Omron CX-Programmer project NewProject (CX-Programmer 9.61)

# PLC NewPLC1: CP1E N30

## Global symbols (name address type ; comment)
0.00 BOOL  ; PB1
0.01 BOOL  ; LS1
0.02 BOOL  ; PS1
0.03 BOOL  ; SS1
0.04 BOOL  ; LS2
0.05 BOOL  ; LS3
0.06 BOOL  ; PB2
0.07 BOOL  ; PB3
0.08 BOOL  ; LS4
100.00 BOOL  ; CR1
100.01 BOOL  ; PL1
100.02 BOOL  ; SOLA
100.03 BOOL  ; CR2
100.04 BOOL  ; SOLB
100.05 BOOL  ; SOLC
100.06 BOOL  ; CR3
100.07 BOOL  ; PL2

## Program NewProgram1 (cyclic task 0)

### Section Section1

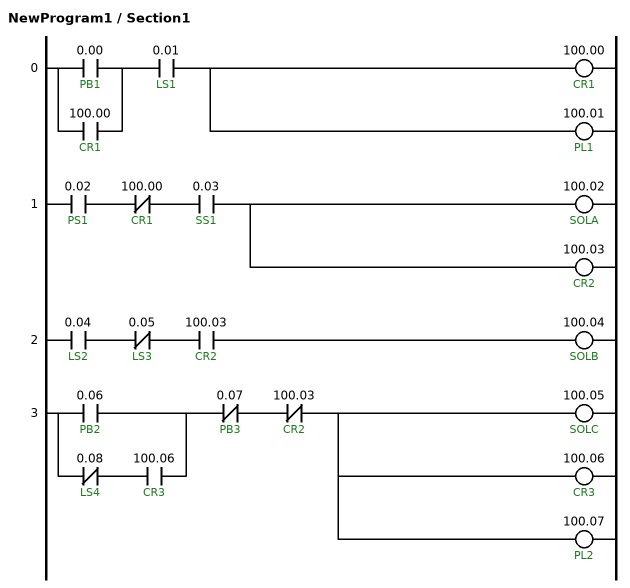
; rung 0
LD 0.00  ; PB1
OR 100.00  ; CR1
AND 0.01  ; LS1
OUT 100.00  ; CR1
OUT 100.01  ; PL1
; rung 1
LD 0.02  ; PS1
ANDNOT 100.00  ; CR1
AND 0.03  ; SS1
OUT 100.02  ; SOLA
OUT 100.03  ; CR2
; rung 2
LD 0.04  ; LS2
ANDNOT 0.05  ; LS3
AND 100.03  ; CR2
OUT 100.04  ; SOLB
; rung 3
LD 0.06  ; PB2
LDNOT 0.08  ; LS4
AND 100.06  ; CR3
ORLD
ANDNOT 0.07  ; PB3
ANDNOT 100.03  ; CR2
OUT 100.05  ; SOLC
OUT 100.06  ; CR3
OUT 100.07  ; PL2

### Section END
; rung 0
END(001)